INTERFACE I_Mode EXTENDS I_Base

METHOD ChangeMode
VAR_INPUT
	RequestedMode : DINT;
END_VAR
END_METHOD

{attribute 'monitoring' := 'call'}
PROPERTY CurrentMode : DINT
GET
END_GET
END_PROPERTY

END_INTERFACE

(* stored: Version 1.1.0.1, ProductVersion 3.1.4026.18
   Itf I_Mode: Id {ad5f09ad-4b02-4231-b384-ecccdfe8b047}
   Method ChangeMode: Id {dd8950ac-e277-45b6-b2ac-81910436f365}
   Property CurrentMode: Id {9ebe5251-c461-45ef-843d-121783cb5fc7}
   Get Get: Id {d643b70e-3ae4-45a6-8188-c439efe9f686} *)
